// TIA Portal V17 export
// export: Created 2024-08-07T21:43:51.7622752Z, ExportSetting WithDefaults, DisplayName Totally Integrated Automation Portal, DisplayVersion V17 Update 7, DisplayName TIA Portal Openness, DisplayVersion V17 Update 7, DisplayName TIA Portal Version Control Interface, DisplayVersion V17, DisplayName SINAMICS Startdrive Advanced, DisplayVersion V17 SP2, DisplayName SINAMICS Startdrive G110M, G120, G120C, G120D, G120P, G115D, DisplayVersion V17 SP2, DisplayName SINAMICS Startdrive G130, G150, S120, S150, SINAMICS MV, S210, DisplayVersion V17 SP2, DisplayName STEP 7 Professional, DisplayVersion V17 Update 7, DisplayName STEP 7 Safety, DisplayVersion V17 Update 6, DisplayName WinCC Advanced / Unified PC, DisplayVersion V17 Update 7
DATA_BLOCK "AnalogControl_DB"   // DB3
VERSION : 0.1
// stored: AutoNumber true, DBAccessibleFromOPCUA true, DBAccessibleFromWebserver true, InstanceOfName AnalogControl, InstanceOfType FB
"AnalogControl"
   // VAR_INPUT
   //    EditIndex : Int := 4;
   //    EditIndexOutput : Int := 1;
   // END_VAR
   // VAR_IN_OUT
   //    save : Bool := FALSE;
   //    load : Bool := FALSE;
   //    saveOutput : Bool := FALSE;
   //    loadOutput : Bool := FALSE;
   // END_VAR
   // VAR
   //    AnalogInputs { S7_SetPoint := 'True'} : Array[1..12] of "AnalogInput";
   //    Inputs { S7_SetPoint := 'True'} : Array[1..12] of Int;
   //    edit : Int := 1;
   //    editedItem : "AnalogInput";
   //    AnalogOutputs { S7_SetPoint := 'True'} : Array[1..12] of "AnalogOutput";
   //    editedItemOutput { S7_SetPoint := 'True'} : "AnalogOutput";
   // END_VAR
BEGIN
   AnalogInputs[1..2].RawValue := 0;
   AnalogInputs[3].RawValue := 2679;
   AnalogInputs[4].RawValue := 2146;
   AnalogInputs[5].RawValue := 32767;
   AnalogInputs[6].RawValue := 0;
   AnalogInputs[7..8].RawValue := 32767;
   AnalogInputs[9..12].RawValue := 0;
   AnalogInputs[1..2].ActualValue := 0.0;
   AnalogInputs[3].ActualValue := 5.813802;
   AnalogInputs[4].ActualValue := 4.657118;
   AnalogInputs[5].ActualValue := 3.051758E-05;
   AnalogInputs[6].ActualValue := 132.6114;
   AnalogInputs[7].ActualValue := 3.814697E-05;
   AnalogInputs[8].ActualValue := -3.814697E-05;
   AnalogInputs[9..12].ActualValue := 0.0;
   AnalogInputs[1..12].ActualValueL := 16#0000;
   AnalogInputs[1..12].MeasurePointA := FALSE;
   AnalogInputs[1..12].MeasurePointB := FALSE;
   AnalogInputs[1..12].Count := FALSE;
   AnalogInputs[1..4].valueA := 0.0;
   AnalogInputs[5].valueA := 32767.0;
   AnalogInputs[6].valueA := 32572.0;
   AnalogInputs[7..8].valueA := 32767.0;
   AnalogInputs[9..12].valueA := 0.0;
   AnalogInputs[1..4].valueB := 27648.0;
   AnalogInputs[5].valueB := 8632.0;
   AnalogInputs[6].valueB := 8010.0;
   AnalogInputs[7].valueB := 6596.0;
   AnalogInputs[8].valueB := 6616.0;
   AnalogInputs[9..12].valueB := 0.0;
   AnalogInputs[1..12].CalibValueA := 0.0;
   AnalogInputs[1..2].CalibValueB := 80.0;
   AnalogInputs[3..4].CalibValueB := 60.0;
   AnalogInputs[5..8].CalibValueB := 100.0;
   AnalogInputs[9..12].CalibValueB := 0.0;
   AnalogInputs[1..2].k := 0.002893518;
   AnalogInputs[3..4].k := 0.002170139;
   AnalogInputs[5].k := -0.00414336;
   AnalogInputs[6].k := -0.00407133;
   AnalogInputs[7].k := -0.003821023;
   AnalogInputs[8].k := -0.003823946;
   AnalogInputs[9..12].k := 1.0;
   AnalogInputs[1..4].c := 0.0;
   AnalogInputs[5].c := 135.7655;
   AnalogInputs[6].c := 132.6114;
   AnalogInputs[7].c := 125.2035;
   AnalogInputs[8].c := 125.2992;
   AnalogInputs[9..12].c := 0.0;
   Inputs[1..2] := 0;
   Inputs[3..4] := 13824;
   Inputs[5] := 3594;
   Inputs[6..12] := 0;
   editedItem.RawValue := 2146;
   editedItem.ActualValue := 4.657118;
   editedItem.ActualValueL := 16#0000;
   editedItem.MeasurePointA := FALSE;
   editedItem.MeasurePointB := FALSE;
   editedItem.Count := FALSE;
   editedItem.valueA := 0.0;
   editedItem.valueB := 27648.0;
   editedItem.CalibValueA := 0.0;
   editedItem.CalibValueB := 60.0;
   editedItem.k := 0.002170139;
   editedItem.c := 0.0;
   AnalogOutputs[1..4].ActualValue := 0.0;
   AnalogOutputs[5].ActualValue := 20.0;
   AnalogOutputs[6..12].ActualValue := 0.0;
   AnalogOutputs[1..2].RawValue := 0;
   AnalogOutputs[3..4].RawValue := 13824;
   AnalogOutputs[5].RawValue := 14376;
   AnalogOutputs[6..12].RawValue := 0;
   AnalogOutputs[1..12].MeasurePointA := FALSE;
   AnalogOutputs[1..12].MeasurePointB := FALSE;
   AnalogOutputs[1..12].Count := FALSE;
   AnalogOutputs[1..3].valueA := -100.0;
   AnalogOutputs[4].valueA := 100.0;
   AnalogOutputs[5..12].valueA := 0.0;
   AnalogOutputs[1..3].valueB := 100.0;
   AnalogOutputs[4].valueB := -100.0;
   AnalogOutputs[5..8].valueB := 100.0;
   AnalogOutputs[9..12].valueB := 0.0;
   AnalogOutputs[1..2].CalibValueA := -27647.0;
   AnalogOutputs[3..12].CalibValueA := 0.0;
   AnalogOutputs[1..2].CalibValueB := 27647.0;
   AnalogOutputs[3..4].CalibValueB := 27648.0;
   AnalogOutputs[5].CalibValueB := 17970.0;
   AnalogOutputs[6].CalibValueB := 27648.0;
   AnalogOutputs[7..8].CalibValueB := 32535.0;
   AnalogOutputs[9..12].CalibValueB := 0.0;
   AnalogOutputs[1..2].k := 276.47;
   AnalogOutputs[3].k := 138.24;
   AnalogOutputs[4].k := -138.24;
   AnalogOutputs[5].k := 179.7;
   AnalogOutputs[6].k := 276.48;
   AnalogOutputs[7..8].k := 325.35;
   AnalogOutputs[9..12].k := 0.0;
   AnalogOutputs[1..2].c := 0.0;
   AnalogOutputs[3..4].c := 13824.0;
   AnalogOutputs[5..12].c := 0.0;
   editedItemOutput.ActualValue := 0.0;
   editedItemOutput.RawValue := 0;
   editedItemOutput.MeasurePointA := FALSE;
   editedItemOutput.MeasurePointB := FALSE;
   editedItemOutput.Count := FALSE;
   editedItemOutput.valueA := -100.0;
   editedItemOutput.valueB := 100.0;
   editedItemOutput.CalibValueA := -27647.0;
   editedItemOutput.CalibValueB := 27647.0;
   editedItemOutput.k := 276.47;
   editedItemOutput.c := 0.0;
END_DATA_BLOCK
